{attribute 'linkalways'} 
{attribute 'no_explicit_call' := 'This FB is a CLASS and must be accessed using methods or properties'}
{attribute 'enable_dynamic_creation'}
FUNCTION_BLOCK FINAL NOT_UINT EXTENDS Node
VAR
	in : _UINT(0);
	out : _UINT(0);
END_VAR

METHOD PUBLIC Clone : I_Node
VAR
	pNode : POINTER TO NOT_UINT;
END_VAR
pNode := __NEW(NOT_UINT);
Clone := pNode^;
END_METHOD

METHOD FB_init : BOOL
VAR_INPUT
	bInitRetains : BOOL; // if TRUE, the retain variables are initialized (warm start / cold start)
	bInCopyCode : BOOL;  // if TRUE, the instance afterwards gets moved into the copy code (online change)
END_VAR
AddInput('in',THIS^.in);
AddOutput('out', THIS^.out);
END_METHOD

METHOD PROTECTED OnExecute
VAR
END_VAR
out.Value := NOT in.Value;
END_METHOD

END_FUNCTION_BLOCK

(* stored: Version 1.1.0.1, ProductVersion 3.1.4024.15
   POU NOT_UINT: Id {fb112558-3560-45ac-a55c-33cc580b7646}, SpecialFunc None
   Folder Constructor: Id {622f60fe-a599-4fb0-89c8-1b9ff498196e}
   Method Clone: Id {56b43048-629c-4215-b3e5-5b6d894e005f}
   Method FB_init: Id {8ab0d29a-6307-4ab4-b39c-e3a613117174}
   Method OnExecute: Id {3635133a-c753-4601-8020-1eb012a70c55} *)
